PROGRAM StateProgram
VAR
	
	Stepper1				: StepperAxis;
	Servo1					: ServoAxis;
	DC1						: DCAxis;
	AxisControlManager		: AxisControlManager;
	
	iAxesManagerCycle		: ITF_CyclicUpdate := AxisControlManager;
	iAxesIndividualCycle	: ARRAY [0..2] OF ITF_CyclicUpdate := [Stepper1, Servo1, DC1];
	
	Result					: HRESULT;
	i						: INT;
	State					: INT;
	
END_VAR


// Switch between the targetted axes AFTER axis functionality has finished
// Prevents switching mid-movement

FOR i := 0 TO 1 BY 1 DO
	iAxesIndividualCycle[i].CyclicUpdate();
END_FOR

Result := iAxesManagerCycle.CyclicUpdate();

CASE State OF
	
	0:
		State := 0;
	
	1:
		AxisControlManager.TargetAxis := Stepper1;
		IF Result = 1 THEN
			State := 0;
		END_IF
		
	2:
		AxisControlManager.TargetAxis := Servo1;
		IF Result = 1 THEN
			State := 0;
		END_IF
		
	3:
		AxisControlManager.TargetAxis := DC1;
		IF Result = 1 THEN
			State := 0;
		END_IF
	
END_CASE

END_PROGRAM

(* stored: Version 1.1.0.1, ProductVersion 3.1.4024.12
   POU StateProgram: Id {1dd6e39d-4307-4e01-a167-86f020bc856f}, SpecialFunc None *)
